{attribute 'GeneratedUsingTerminal: EL3312-0000-0016'}
{attribute addProperty BoxType "EL3312-0000-0016"}
{attribute addProperty Description "EL3312 2Ch. Ana. Input Thermocouple (TC)"}
{attribute addProperty Physics "KK"}
{attribute addProperty Id "TC_Inputs_Channel_1AT %I*TC_Inputs_Channel_EA9DF21E9TC_Inputs_Channel_2AT %I*TC_Inputs_Channel_EA9DF21E9WcStateAT %I*WcState_9091E0EB2InfoDataAT %I*InfoData_32EB74EA10"}
{attribute addProperty CRC "1214600323"}
{attribute addProperty Size "30"}
TYPE EL3312_48655483 EXTENDS EtcSlaveTerminalBase_947E5A46 :
STRUCT
	{attribute addProperty Name "TC_Inputs_Channel_1"}
	TC_Inputs_Channel_1 : TC_Inputs_Channel_EA9DF21E;
	{attribute addProperty Name "TC_Inputs_Channel_2"}
	TC_Inputs_Channel_2 : TC_Inputs_Channel_EA9DF21E;
	{attribute addProperty Name "WcState"}
	WcState : WcState_9091E0EB;
	{attribute addProperty Name "InfoData"}
	InfoData : InfoData_32EB74EA;
END_STRUCT
END_TYPE

(* stored: Version 1.2.0.0, ProductVersion 3.1.4024.11
   DUT EL3312_48655483: Id {c7bad529-adce-4ede-b6de-3200f192cfd0} *)
